FUNCTION_BLOCK FB_BacklashCompensationNC IMPLEMENTS I_BacklashCompensation
VAR_INPUT
END_VAR
VAR_OUTPUT
END_VAR
VAR
(* Other status information for users of the IOC *)
    (* Backlash compensation*)
    // Enabled axis backlash compensation
    {attribute 'pytmc' := '
        pv: PLC:bBacklashCompUserEn
        io: io
        field: ZNAM FALSE
        field: ONAM TRUE
        field: DESC Enable Backlash compensation
    '}
    bUserEnable: BOOL;

    // backlash compensation status
    {attribute 'pytmc' := '
        pv: PLC:bBacklashCompStatus
        io: i
        field: ZNAM DISABLED
        field: ONAM ENABLED
        field: DESC Backlash compensation status
    '}
    bBacklashCompStatus: BOOL;

    // Backlash compensation value
    {attribute 'pytmc' := '
        pv: PLC:fBacklashComp
        io: io
        field: DESC Backlash compensation
    '}
    fBacklashComp: LREAL := 0.0;

    // Current Backlash compensation value ?
    {attribute 'pytmc' := '
        pv: PLC:fMeasuredBacklashComp
        io: i
        field: DESC Currently applied compensation
    '}
    fActCompensation: LREAL;

    {attribute 'no_copy'}
    AxisRef : REFERENCE TO AXIS_REF;
    fbMcBacklashCompensation: MC_BacklashCompensation;
    fPrevCompensation : LREAL := 0.0;
    bActive: BOOL;
    fRampVelo : LREAL := 0.0;
    bLocalEnable : BOOL;
    bError : BOOL;
    bBusy : BOOL;
    nErrorID : UDINT;
    sMessage : T_MAXSTRING;
    eDisableMode: E_DisableMode := E_DISABLEMODE.DisableModeHold;

END_VAR

PROPERTY Aborted : BOOL
GET
END_GET
END_PROPERTY

PROPERTY ActCompensation : LREAL
GET
ActCompensation := fActCompensation;
END_GET
END_PROPERTY

PROPERTY Active : BOOL
GET
Active:=fbMcBacklashCompensation.Enabled;
END_GET
END_PROPERTY

(*
    Handle positive/negative backlash compensation
    User needs to set the direction of backlash from the sign of the compensation value
    Backlash compensation is disabled during referencing (homing).
    When direction is positive/negative, further movement in the negative/positive direction not compensated
    further movement in the negative/positive direction will be compensated
*)
METHOD BacklashCompensation
VAR_INPUT
    Activate     : BOOL;
    Compensation	: LREAL;
    RampVelocity	: LREAL;
    DisableMode	: E_DISABLEMODE := E_DISABLEMODE.DisableModeHold;
END_VAR
THIS^.bActive:= Activate;
THIS^.fBacklashComp := Compensation;
THIS^.fRampVelo := RampVelocity;
THIS^.eDisableMode:=DisableMode;
END_METHOD

(*synced Fbs need just to activate the compensation with a given ramp speed
  other parameters are provided via EPICS (declared in this FB) or via the more extended BackalshCompensation method (simulation) *)
METHOD BacklashCompensationActive
VAR_INPUT
    Active	: BOOL;
    RampVelocity	: LREAL;
END_VAR
THIS^.bActive:= Active;
THIS^.fRampVelo := RampVelocity;
END_METHOD

PROPERTY Busy : BOOL
GET
Busy := fbMcBacklashCompensation.Busy;
END_GET
END_PROPERTY

METHOD PUBLIC CallAfterInit
VAR_INPUT
    AxisRef : REFERENCE TO AXIS_REF;
END_VAR
THIS^.AxisRef REF= AxisRef;
END_METHOD

PROPERTY Done : BOOL
GET
END_GET
END_PROPERTY

PROPERTY Error : BOOL
GET
Error := THIS^.bError;
END_GET
END_PROPERTY

PROPERTY ErrorID : UDINT
GET
ErrorID := THIS^.nErrorID;
END_GET
END_PROPERTY

METHOD FB_Init : BOOL
VAR_INPUT
    bInitRetains : BOOL; // if TRUE, the retain variables are initialized (warm start / cold start)
    bInCopyCode : BOOL;  // if TRUE, the instance afterwards gets moved into the copy code (online change)
    AxisRef : REFERENCE TO AXIS_REF;
END_VAR
THIS^.AxisRef REF= AxisRef;
END_METHOD

PROPERTY Message : T_MaxString
GET
Message :=sMessage;
END_GET
END_PROPERTY

PROPERTY UserEnable : BOOL
SET
bUserEnable := UserEnable;
END_SET
END_PROPERTY

END_FUNCTION_BLOCK

(* stored: Version 1.1.0.1
   POU FB_BacklashCompensationNC: Id {15421978-726d-43ca-8e30-d33510c30e01}, SpecialFunc None
   Property Aborted: Id {59820488-53e0-4bd0-9746-41b9b903c795}
   Get Get: Id {af423ed0-d781-4de7-b003-71fdc1e2f7f8}
   Property ActCompensation: Id {022a8867-c28c-4e7c-88fa-1c1e1f6f1ad1}
   Get Get: Id {bb138911-4f3b-47a1-847c-b5cced113ef6}
   Property Active: Id {fa202a56-38e3-4b3a-bf52-57135d76cf34}
   Get Get: Id {08ef6077-f2d4-42e4-90da-6c52adfa9a0a}
   Method BacklashCompensation: Id {28619ab5-da60-4dc4-96a8-3e2ae3773706}
   Method BacklashCompensationActive: Id {dbabc34f-4a46-42a1-a3aa-48ed4e21c0cc}
   Property Busy: Id {55ee7371-1408-415b-b1f0-122aa6241483}
   Get Get: Id {7637bb84-185d-4e7a-b993-3057df36bf56}
   Method CallAfterInit: Id {59b21a6b-3d1b-46f2-866a-5384398ac207}
   Property Done: Id {aa40d0fa-7dfa-4048-b1f0-b1c583de1e82}
   Get Get: Id {9933535c-b83d-458a-8f5e-e58dec905ec5}
   Property Error: Id {0213434a-d40a-49c7-a6b4-a3e9e9a7a41a}
   Get Get: Id {c1a3c97c-ae91-4276-85b5-feecf9e8d7c5}
   Property ErrorID: Id {b6765fc0-40e7-4ce5-aa13-569ea50920db}
   Get Get: Id {3dbdc77e-7172-4e8a-b541-0b84a6087295}
   Method FB_Init: Id {86eeb26b-dd4d-42ae-bdf4-cda3d947fa1b}
   Property Message: Id {799861dc-10f6-42dd-a8b5-747f46787023}
   Get Get: Id {b04d60be-1e7a-4ed8-aad3-cee013905d08}
   Property UserEnable: Id {a9d2d8cc-e94d-4db5-bf54-daa67dbaf501}
   Set Set: Id {2cefc03c-c62d-4e89-aa15-5c5cbbb4411a} *)
